% RSLogix 500 project Programa Respirador.RSS, saved by version 8.30.00.16 %
PROJECT "UNTITLED"    % processor: Bul.1763 MicroLogix 1100 Series B %

PROGRAM FILES
  LAD 2   9 rungs

DATA FILES
  O0 OUTPUT  4 elements
  I1 INPUT  6 elements
  S2 STATUS  66 elements
  B3 BINARY  1 elements
  T4 TIMER  2 elements
  C5 COUNTER  1 elements
  R6 CONTROL  1 elements
  N7 INTEGER  2 elements
  F8 FLOAT  1 elements

LADDER 2
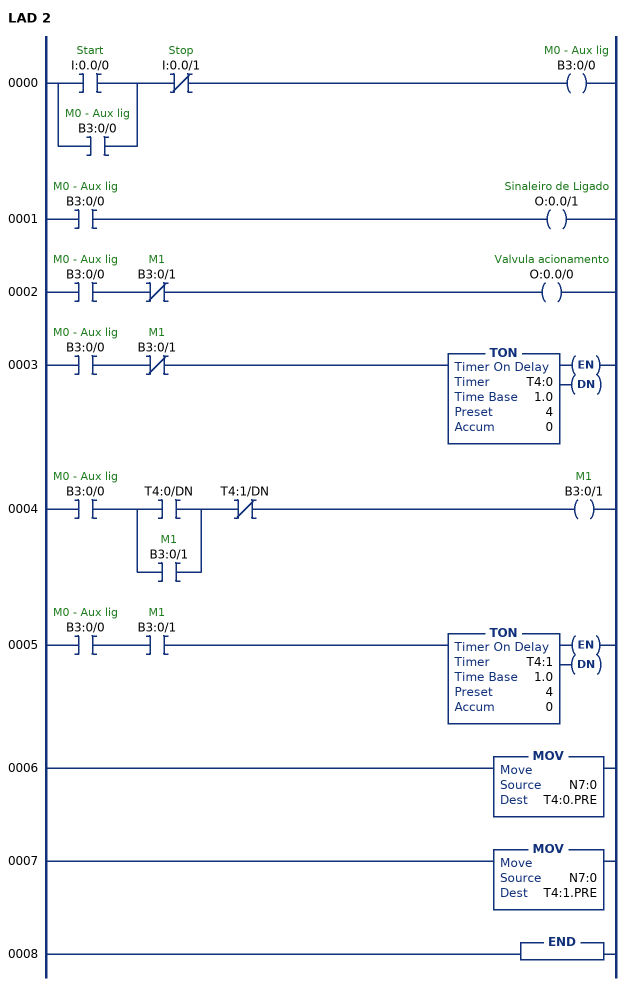
% Rung: 0 %
SOR BST XIC I:0.0/0 NXB XIC B3:0/0 BND XIO I:0.0/1 OTE B3:0/0 EOR
%   I:0.0/0  "Start" %
%   B3:0/0  "M0 - Aux lig" %
%   I:0.0/1  "Stop" %
% Rung: 1 %
SOR XIC B3:0/0 OTE O:0.0/1 EOR
%   B3:0/0  "M0 - Aux lig" %
%   O:0.0/1  "Sinaleiro de Ligado" %
% Rung: 2 %
SOR XIC B3:0/0 XIO B3:0/1 OTE O:0.0/0 EOR
%   B3:0/0  "M0 - Aux lig" %
%   B3:0/1  "M1" %
%   O:0.0/0  "Valvula acionamento" %
% Rung: 3 %
SOR XIC B3:0/0 XIO B3:0/1 TON T4:0 1.0 4 0 EOR
%   B3:0/0  "M0 - Aux lig" %
%   B3:0/1  "M1" %
% Rung: 4 %
SOR XIC B3:0/0 BST XIC T4:0/DN NXB XIC B3:0/1 BND XIO T4:1/DN OTE B3:0/1 EOR
%   B3:0/0  "M0 - Aux lig" %
%   B3:0/1  "M1" %
% Rung: 5 %
SOR XIC B3:0/0 XIC B3:0/1 TON T4:1 1.0 4 0 EOR
%   B3:0/0  "M0 - Aux lig" %
%   B3:0/1  "M1" %
% Rung: 6 %
SOR MOV N7:0 T4:0.PRE EOR
% Rung: 7 %
SOR MOV N7:0 T4:1.PRE EOR
% Rung: 8 %
SOR END EOR

OTHER DOCUMENTED ADDRESSES
  B1:0/0  "M1"
  START  "O.O/0"

DATA TABLE (non-zero values as saved)
DATA T4
% .PRE .ACC %
% T4:0 % 4 0
% T4:1 % 4 0
DATA N7
% N7:0 % 4 0
